FUNCTION FUNC_NoReturn
VAR_INPUT
  nInput : INT;
END_VAR

;

END_FUNCTION

(* stored: Version 1.1.0.1, ProductVersion 3.1.4024.12
   POU FUNC_NoReturn: Id {f1a2b3c4-d5e6-7890-abcd-ef1234567895}, SpecialFunc None *)
